TYPE E_DilType :
(
	DILTYPE_Single := 0,
	DILTYPE_TwinParallel := 1,
	DILTYPE_TwinSerial := 2,
	DILTYPE_TwinTransfer := 3
)USINT;
END_TYPE

(* stored: Version 1.1.0.1, ProductVersion 3.1.0.25
   DUT E_DilType: Id {39f8dde6-590b-4cfb-af55-67ab2e211db4} *)
